// TIA Portal V18 export
FUNCTION "SS2_A2_8AO_IO_Update" : Void   // FC11130, LAD
{ S7_Optimized_Access := 'TRUE' }
VERSION : 0.1
// stored: AutoNumber false, IsIECCheckEnabled false, SetENOAutomatically false, UDAEnableTagReadback false
BEGIN

REGION Network 1: AO0
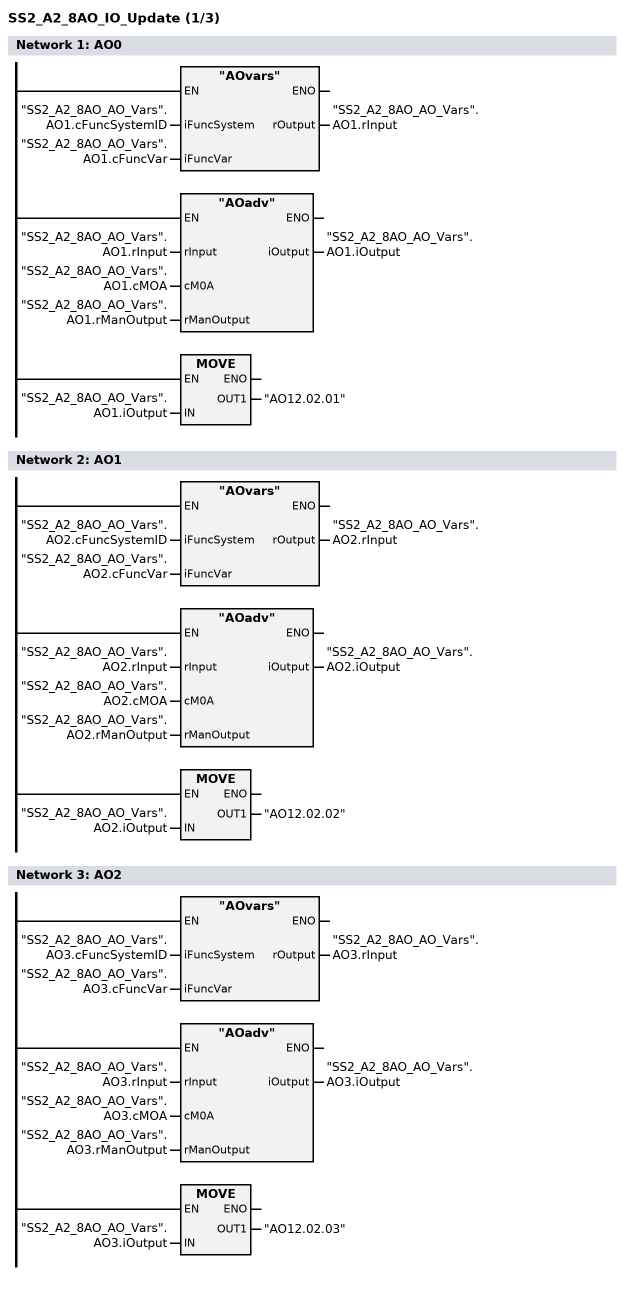
   RUNG wire#powerrail
      "AOvars"(iFuncSystem := "SS2_A2_8AO_AO_Vars".AO1.cFuncSystemID, iFuncVar := "SS2_A2_8AO_AO_Vars".AO1.cFuncVar, rOutput => "SS2_A2_8AO_AO_Vars".AO1.rInput)
   END_RUNG
   RUNG wire#powerrail
      "AOadv"(rInput := "SS2_A2_8AO_AO_Vars".AO1.rInput, cM0A := "SS2_A2_8AO_AO_Vars".AO1.cMOA, rManOutput := "SS2_A2_8AO_AO_Vars".AO1.rManOutput, iOutput => "SS2_A2_8AO_AO_Vars".AO1.iOutput)
   END_RUNG
   RUNG wire#powerrail
      Move(in := "SS2_A2_8AO_AO_Vars".AO1.iOutput, out1 => "AO12.02.01")
   END_RUNG
   // the same network as SCL:
   "AOvars"(iFuncSystem := "SS2_A2_8AO_AO_Vars".AO1.cFuncSystemID,
            iFuncVar := "SS2_A2_8AO_AO_Vars".AO1.cFuncVar,
            rOutput => "SS2_A2_8AO_AO_Vars".AO1.rInput);
   "AOadv"(rInput := "SS2_A2_8AO_AO_Vars".AO1.rInput,
           cM0A := "SS2_A2_8AO_AO_Vars".AO1.cMOA,
           rManOutput := "SS2_A2_8AO_AO_Vars".AO1.rManOutput,
           iOutput => "SS2_A2_8AO_AO_Vars".AO1.iOutput);
   "AO12.02.01" := "SS2_A2_8AO_AO_Vars".AO1.iOutput;
END_REGION

REGION Network 2: AO1
   RUNG wire#powerrail
      "AOvars"(iFuncSystem := "SS2_A2_8AO_AO_Vars".AO2.cFuncSystemID, iFuncVar := "SS2_A2_8AO_AO_Vars".AO2.cFuncVar, rOutput => "SS2_A2_8AO_AO_Vars".AO2.rInput)
   END_RUNG
   RUNG wire#powerrail
      "AOadv"(rInput := "SS2_A2_8AO_AO_Vars".AO2.rInput, cM0A := "SS2_A2_8AO_AO_Vars".AO2.cMOA, rManOutput := "SS2_A2_8AO_AO_Vars".AO2.rManOutput, iOutput => "SS2_A2_8AO_AO_Vars".AO2.iOutput)
   END_RUNG
   RUNG wire#powerrail
      Move(in := "SS2_A2_8AO_AO_Vars".AO2.iOutput, out1 => "AO12.02.02")
   END_RUNG
   // the same network as SCL:
   "AOvars"(iFuncSystem := "SS2_A2_8AO_AO_Vars".AO2.cFuncSystemID,
            iFuncVar := "SS2_A2_8AO_AO_Vars".AO2.cFuncVar,
            rOutput => "SS2_A2_8AO_AO_Vars".AO2.rInput);
   "AOadv"(rInput := "SS2_A2_8AO_AO_Vars".AO2.rInput,
           cM0A := "SS2_A2_8AO_AO_Vars".AO2.cMOA,
           rManOutput := "SS2_A2_8AO_AO_Vars".AO2.rManOutput,
           iOutput => "SS2_A2_8AO_AO_Vars".AO2.iOutput);
   "AO12.02.02" := "SS2_A2_8AO_AO_Vars".AO2.iOutput;
END_REGION

REGION Network 3: AO2
   RUNG wire#powerrail
      "AOvars"(iFuncSystem := "SS2_A2_8AO_AO_Vars".AO3.cFuncSystemID, iFuncVar := "SS2_A2_8AO_AO_Vars".AO3.cFuncVar, rOutput => "SS2_A2_8AO_AO_Vars".AO3.rInput)
   END_RUNG
   RUNG wire#powerrail
      "AOadv"(rInput := "SS2_A2_8AO_AO_Vars".AO3.rInput, cM0A := "SS2_A2_8AO_AO_Vars".AO3.cMOA, rManOutput := "SS2_A2_8AO_AO_Vars".AO3.rManOutput, iOutput => "SS2_A2_8AO_AO_Vars".AO3.iOutput)
   END_RUNG
   RUNG wire#powerrail
      Move(in := "SS2_A2_8AO_AO_Vars".AO3.iOutput, out1 => "AO12.02.03")
   END_RUNG
   // the same network as SCL:
   "AOvars"(iFuncSystem := "SS2_A2_8AO_AO_Vars".AO3.cFuncSystemID,
            iFuncVar := "SS2_A2_8AO_AO_Vars".AO3.cFuncVar,
            rOutput => "SS2_A2_8AO_AO_Vars".AO3.rInput);
   "AOadv"(rInput := "SS2_A2_8AO_AO_Vars".AO3.rInput,
           cM0A := "SS2_A2_8AO_AO_Vars".AO3.cMOA,
           rManOutput := "SS2_A2_8AO_AO_Vars".AO3.rManOutput,
           iOutput => "SS2_A2_8AO_AO_Vars".AO3.iOutput);
   "AO12.02.03" := "SS2_A2_8AO_AO_Vars".AO3.iOutput;
END_REGION

REGION Network 4: AO3
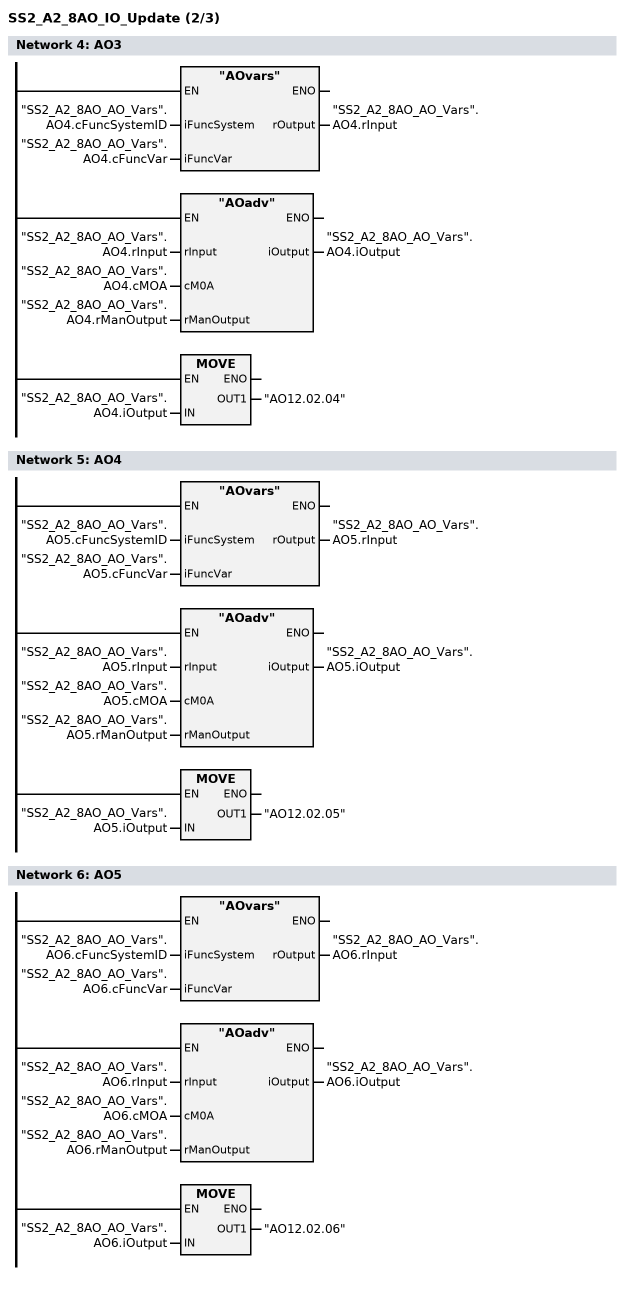
   RUNG wire#powerrail
      "AOvars"(iFuncSystem := "SS2_A2_8AO_AO_Vars".AO4.cFuncSystemID, iFuncVar := "SS2_A2_8AO_AO_Vars".AO4.cFuncVar, rOutput => "SS2_A2_8AO_AO_Vars".AO4.rInput)
   END_RUNG
   RUNG wire#powerrail
      "AOadv"(rInput := "SS2_A2_8AO_AO_Vars".AO4.rInput, cM0A := "SS2_A2_8AO_AO_Vars".AO4.cMOA, rManOutput := "SS2_A2_8AO_AO_Vars".AO4.rManOutput, iOutput => "SS2_A2_8AO_AO_Vars".AO4.iOutput)
   END_RUNG
   RUNG wire#powerrail
      Move(in := "SS2_A2_8AO_AO_Vars".AO4.iOutput, out1 => "AO12.02.04")
   END_RUNG
   // the same network as SCL:
   "AOvars"(iFuncSystem := "SS2_A2_8AO_AO_Vars".AO4.cFuncSystemID,
            iFuncVar := "SS2_A2_8AO_AO_Vars".AO4.cFuncVar,
            rOutput => "SS2_A2_8AO_AO_Vars".AO4.rInput);
   "AOadv"(rInput := "SS2_A2_8AO_AO_Vars".AO4.rInput,
           cM0A := "SS2_A2_8AO_AO_Vars".AO4.cMOA,
           rManOutput := "SS2_A2_8AO_AO_Vars".AO4.rManOutput,
           iOutput => "SS2_A2_8AO_AO_Vars".AO4.iOutput);
   "AO12.02.04" := "SS2_A2_8AO_AO_Vars".AO4.iOutput;
END_REGION

REGION Network 5: AO4
   RUNG wire#powerrail
      "AOvars"(iFuncSystem := "SS2_A2_8AO_AO_Vars".AO5.cFuncSystemID, iFuncVar := "SS2_A2_8AO_AO_Vars".AO5.cFuncVar, rOutput => "SS2_A2_8AO_AO_Vars".AO5.rInput)
   END_RUNG
   RUNG wire#powerrail
      "AOadv"(rInput := "SS2_A2_8AO_AO_Vars".AO5.rInput, cM0A := "SS2_A2_8AO_AO_Vars".AO5.cMOA, rManOutput := "SS2_A2_8AO_AO_Vars".AO5.rManOutput, iOutput => "SS2_A2_8AO_AO_Vars".AO5.iOutput)
   END_RUNG
   RUNG wire#powerrail
      Move(in := "SS2_A2_8AO_AO_Vars".AO5.iOutput, out1 => "AO12.02.05")
   END_RUNG
   // the same network as SCL:
   "AOvars"(iFuncSystem := "SS2_A2_8AO_AO_Vars".AO5.cFuncSystemID,
            iFuncVar := "SS2_A2_8AO_AO_Vars".AO5.cFuncVar,
            rOutput => "SS2_A2_8AO_AO_Vars".AO5.rInput);
   "AOadv"(rInput := "SS2_A2_8AO_AO_Vars".AO5.rInput,
           cM0A := "SS2_A2_8AO_AO_Vars".AO5.cMOA,
           rManOutput := "SS2_A2_8AO_AO_Vars".AO5.rManOutput,
           iOutput => "SS2_A2_8AO_AO_Vars".AO5.iOutput);
   "AO12.02.05" := "SS2_A2_8AO_AO_Vars".AO5.iOutput;
END_REGION

REGION Network 6: AO5
   RUNG wire#powerrail
      "AOvars"(iFuncSystem := "SS2_A2_8AO_AO_Vars".AO6.cFuncSystemID, iFuncVar := "SS2_A2_8AO_AO_Vars".AO6.cFuncVar, rOutput => "SS2_A2_8AO_AO_Vars".AO6.rInput)
   END_RUNG
   RUNG wire#powerrail
      "AOadv"(rInput := "SS2_A2_8AO_AO_Vars".AO6.rInput, cM0A := "SS2_A2_8AO_AO_Vars".AO6.cMOA, rManOutput := "SS2_A2_8AO_AO_Vars".AO6.rManOutput, iOutput => "SS2_A2_8AO_AO_Vars".AO6.iOutput)
   END_RUNG
   RUNG wire#powerrail
      Move(in := "SS2_A2_8AO_AO_Vars".AO6.iOutput, out1 => "AO12.02.06")
   END_RUNG
   // the same network as SCL:
   "AOvars"(iFuncSystem := "SS2_A2_8AO_AO_Vars".AO6.cFuncSystemID,
            iFuncVar := "SS2_A2_8AO_AO_Vars".AO6.cFuncVar,
            rOutput => "SS2_A2_8AO_AO_Vars".AO6.rInput);
   "AOadv"(rInput := "SS2_A2_8AO_AO_Vars".AO6.rInput,
           cM0A := "SS2_A2_8AO_AO_Vars".AO6.cMOA,
           rManOutput := "SS2_A2_8AO_AO_Vars".AO6.rManOutput,
           iOutput => "SS2_A2_8AO_AO_Vars".AO6.iOutput);
   "AO12.02.06" := "SS2_A2_8AO_AO_Vars".AO6.iOutput;
END_REGION

REGION Network 7: AO6
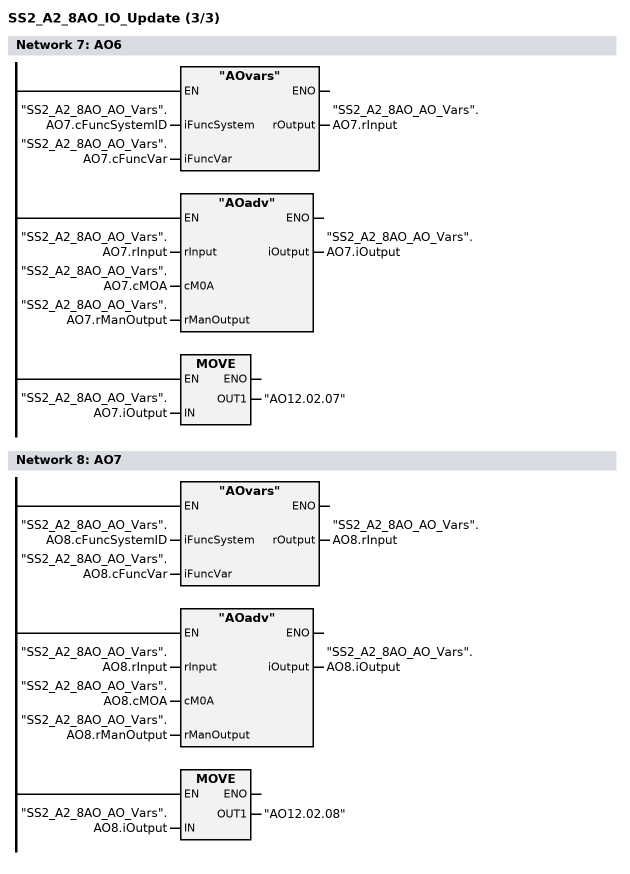
   RUNG wire#powerrail
      "AOvars"(iFuncSystem := "SS2_A2_8AO_AO_Vars".AO7.cFuncSystemID, iFuncVar := "SS2_A2_8AO_AO_Vars".AO7.cFuncVar, rOutput => "SS2_A2_8AO_AO_Vars".AO7.rInput)
   END_RUNG
   RUNG wire#powerrail
      "AOadv"(rInput := "SS2_A2_8AO_AO_Vars".AO7.rInput, cM0A := "SS2_A2_8AO_AO_Vars".AO7.cMOA, rManOutput := "SS2_A2_8AO_AO_Vars".AO7.rManOutput, iOutput => "SS2_A2_8AO_AO_Vars".AO7.iOutput)
   END_RUNG
   RUNG wire#powerrail
      Move(in := "SS2_A2_8AO_AO_Vars".AO7.iOutput, out1 => "AO12.02.07")
   END_RUNG
   // the same network as SCL:
   "AOvars"(iFuncSystem := "SS2_A2_8AO_AO_Vars".AO7.cFuncSystemID,
            iFuncVar := "SS2_A2_8AO_AO_Vars".AO7.cFuncVar,
            rOutput => "SS2_A2_8AO_AO_Vars".AO7.rInput);
   "AOadv"(rInput := "SS2_A2_8AO_AO_Vars".AO7.rInput,
           cM0A := "SS2_A2_8AO_AO_Vars".AO7.cMOA,
           rManOutput := "SS2_A2_8AO_AO_Vars".AO7.rManOutput,
           iOutput => "SS2_A2_8AO_AO_Vars".AO7.iOutput);
   "AO12.02.07" := "SS2_A2_8AO_AO_Vars".AO7.iOutput;
END_REGION

REGION Network 8: AO7
   RUNG wire#powerrail
      "AOvars"(iFuncSystem := "SS2_A2_8AO_AO_Vars".AO8.cFuncSystemID, iFuncVar := "SS2_A2_8AO_AO_Vars".AO8.cFuncVar, rOutput => "SS2_A2_8AO_AO_Vars".AO8.rInput)
   END_RUNG
   RUNG wire#powerrail
      "AOadv"(rInput := "SS2_A2_8AO_AO_Vars".AO8.rInput, cM0A := "SS2_A2_8AO_AO_Vars".AO8.cMOA, rManOutput := "SS2_A2_8AO_AO_Vars".AO8.rManOutput, iOutput => "SS2_A2_8AO_AO_Vars".AO8.iOutput)
   END_RUNG
   RUNG wire#powerrail
      Move(in := "SS2_A2_8AO_AO_Vars".AO8.iOutput, out1 => "AO12.02.08")
   END_RUNG
   // the same network as SCL:
   "AOvars"(iFuncSystem := "SS2_A2_8AO_AO_Vars".AO8.cFuncSystemID,
            iFuncVar := "SS2_A2_8AO_AO_Vars".AO8.cFuncVar,
            rOutput => "SS2_A2_8AO_AO_Vars".AO8.rInput);
   "AOadv"(rInput := "SS2_A2_8AO_AO_Vars".AO8.rInput,
           cM0A := "SS2_A2_8AO_AO_Vars".AO8.cMOA,
           rManOutput := "SS2_A2_8AO_AO_Vars".AO8.rManOutput,
           iOutput => "SS2_A2_8AO_AO_Vars".AO8.iOutput);
   "AO12.02.08" := "SS2_A2_8AO_AO_Vars".AO8.iOutput;
END_REGION
END_FUNCTION
